FUNCTION_BLOCK FB_Service_IOs
VAR_INPUT
END_VAR
VAR_OUTPUT
END_VAR
VAR
END_VAR

END_FUNCTION_BLOCK

(* stored: Version 1.1.0.1, ProductVersion 3.1.4024.12
   POU FB_Service_IOs: Id {db4b2c86-66d8-4aa5-8a6b-26c2bfdd0e13}, SpecialFunc None *)
